{attribute 'qualified_only'}
VAR_GLOBAL
    CELL_RATED_CAPACITY_AmpHours : LREAL := 2.5;
 
    CELLS_PER_MODULE : INT := 16;
END_VAR

(* stored: Version 1.1.0.1
   GVL GVL_BatteryConstants: Id {162ce7a6-0b6f-4610-9e73-e7086941e053} *)
